TYPE ST_Pose :
STRUCT
	x : LREAL;
	y : LREAL;
	z: LREAL;
	roll: LREAL;
	pitch: LREAL;
	yaw: LREAL; //THETA
END_STRUCT
END_TYPE

(* stored: Version 1.1.0.1, ProductVersion 3.1.4026.18
   DUT ST_Pose: Id {e4f90f08-2c74-4a3a-b4af-3a5868a4d9f1} *)
